(* PLC project Unnamed, Unknown Unnamed 1 *)
(* stored: creationDateTime 2025-11-04T16:58:52, modificationDateTime 2025-11-04T17:00:59 *)

PROGRAM main
  VAR
    Trigger : BOOL := False;
    Break : BOOL := False;
    Condition : BOOL := False;
  END_VAR

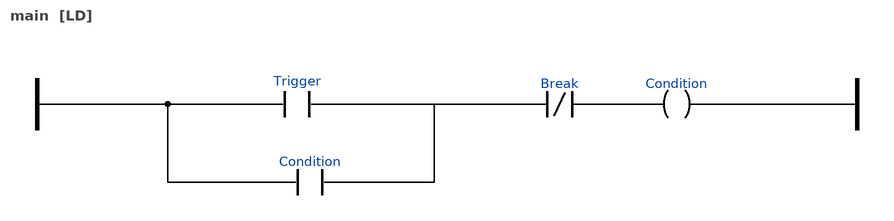
(* LD diagram, written out as Structured Text *)
Condition := (Trigger OR Condition) AND NOT Break;
END_PROGRAM

CONFIGURATION Config0
  RESOURCE Res0 ON PLC
    TASK task0(INTERVAL := T#20ms, PRIORITY := 0);
    PROGRAM instance0 WITH task0 : main;
  END_RESOURCE
END_CONFIGURATION
